// TIA Portal V20 export
DATA_BLOCK "DB_AsiSetpoint"   // DB31
// stored: Access Published, MemoryReserve 100, Namespace ProductionLine
   VAR
      Line : Struct
         ProductionLine : Struct
            DirChange : Struct
               Conveyor : Array[_.minProductionLine.._.maxProductionLine] of Bool;
            END_STRUCT;
            Speed : Struct
               Conveyor : Array[_.minProductionLine.._.maxProductionLine] of Bool;
            END_STRUCT;
         END_STRUCT;
      END_STRUCT;
   END_VAR
BEGIN
   // Line.ProductionLine.DirChange.Conveyor[1001] : AS1.1.1
   // Line.ProductionLine.DirChange.Conveyor[1002] : AS1.1.2
   // Line.ProductionLine.Speed.Conveyor[1001] : AS1.1.1
   // Line.ProductionLine.Speed.Conveyor[1002] : AS1.1.2
END_DATA_BLOCK
